Staubli VAL3: getMean.pgx

public program getMean(num& x_nInput[], num& x_nMean)
  local num l_nCount
  local num l_nSum
begin

  l_nSum = 0

  for l_nCount = 0 to size(x_nInput)-1
    l_nSum = l_nSum + x_nInput[l_nCount]
  endFor

  x_nMean = l_nSum/size(x_nInput)

end
